// TIA Portal project "SelecaoProjeto" (V15)

(* hardware
DEVICE "S7-1200 station_1"  S7-1200 Station
   slot 0: "Rack_0"  S7-1200 Rack  Rack  V1.0
   slot 1: "PLC_1"  CPU 1214C DC/DC/DC  6ES7 214-1AG40-0XB0  V4.2
   slot 2: "DI 8x24VDC_1"  SM 1221 DI8 x 24VDC  6ES7 221-1BF30-0XB0  V1.0
*)

// ===== PLC "PLC_1"  CPU 1214C DC/DC/DC =====

VAR_GLOBAL   // PLC tag table "Default tag table"
   "BtnStop" AT %I0.0 : Bool;
   "BtnStart" AT %I0.1 : Bool;
   "S2Capacitivo" AT %I0.2 : Bool;
   "S1Indutivo" AT %I0.3 : Bool;
   "S3Pequeno" AT %I0.4 : Bool;
   "S4Medio" AT %I0.5 : Bool;
   "S5Grande" AT %I0.6 : Bool;
   "Resetar defeito" AT %I0.7 : Bool;
   "S6_FimDeCurso" AT %I1.0 : Bool;
   "Reed_Switch1" AT %I1.1 : Bool;
   "Reed_Switch2" AT %I1.2 : Bool;
   "Reed_Switch3" AT %I1.3 : Bool;
   "SnOtico_Grande" AT %I1.4 : Bool;
   "SnOtico_Medio" AT %I1.5 : Bool;
   "SnOtico_Pequeno" AT %I8.0 : Bool;
   "Motor1" AT %Q0.1 : Bool;
   "LampadaDefeito" AT %Q0.2 : Bool;
   "Soleoneide1" AT %Q0.3 : Bool;
   "Soleoneide2" AT %Q0.4 : Bool;
   "Soleoneide3" AT %Q0.5 : Bool;
   "SemDefeito1" AT %M0.1 : Bool;
   "SemDefeito2" AT %M0.2 : Bool;
   "MotorPronto" AT %M0.4 : Bool;
   "S1acionado" AT %M0.5 : Bool;
   "S2Acionado" AT %M0.6 : Bool;
   "Metalico" AT %M1.0 : Bool;
   "NaoMetalico" AT %M1.1 : Bool;
   "Vazio" AT %M1.2 : Bool;
   "MotorSetado" AT %M0.7 : Bool;
   "S3Acionado" AT %M1.3 : Bool;
   "S4Acionado" AT %M1.4 : Bool;
   "S5Acionado" AT %M1.5 : Bool;
   "Grande" AT %M2.0 : Bool;
   "Medio" AT %M2.1 : Bool;
   "Pequeno" AT %M2.2 : Bool;
   "Vazio2" AT %M1.7 : Bool;
   "Sistema com defeito" AT %M3.0 : Bool;
   "Zera_Contagem" AT %M0.3 : Bool;
   "Rejeitado" AT %M4.0 : Bool;
   "Solenoide_Recuado" AT %M4.1 : Bool;
   "Contagem_Grande" AT %M4.2 : Bool;
   "Contagem_Media" AT %M4.3 : Bool;
   "Contagem_Pequena" AT %M4.4 : Bool;
END_VAR

// folder: System blocks/Program resources

DATA_BLOCK "IEC_Counter_0_DB"   // DB1
{ S7_Optimized_Access := 'TRUE' }
AUTHOR : Simatic
FAMILY : IEC
NAME : CNTR
VERSION : 1.0
// stored: InstanceOfName IEC_COUNTER
"IEC_COUNTER"
BEGIN
END_DATA_BLOCK

DATA_BLOCK "IEC_Counter_0_DB_2"   // DB3
{ S7_Optimized_Access := 'TRUE' }
AUTHOR : Simatic
FAMILY : IEC
NAME : CNTR
VERSION : 1.0
// stored: InstanceOfName IEC_COUNTER
"IEC_COUNTER"
BEGIN
END_DATA_BLOCK

DATA_BLOCK "IEC_Counter_0_DB_3"   // DB4
{ S7_Optimized_Access := 'TRUE' }
AUTHOR : Simatic
FAMILY : IEC
NAME : CNTR
VERSION : 1.0
// stored: InstanceOfName IEC_COUNTER
"IEC_COUNTER"
BEGIN
END_DATA_BLOCK

DATA_BLOCK "IEC_Counter_0_DB_4"   // DB5
{ S7_Optimized_Access := 'TRUE' }
AUTHOR : Simatic
FAMILY : IEC
NAME : CNTR
VERSION : 1.0
// stored: InstanceOfName IEC_COUNTER
"IEC_COUNTER"
BEGIN
END_DATA_BLOCK

// folder: (top level)

FUNCTION "Selecao" : Void   // FC1, LAD
{ S7_Optimized_Access := 'TRUE' }
VERSION : 0.1
// Projeto Separação de peças
BEGIN

REGION Network 1
   // Setar Motor
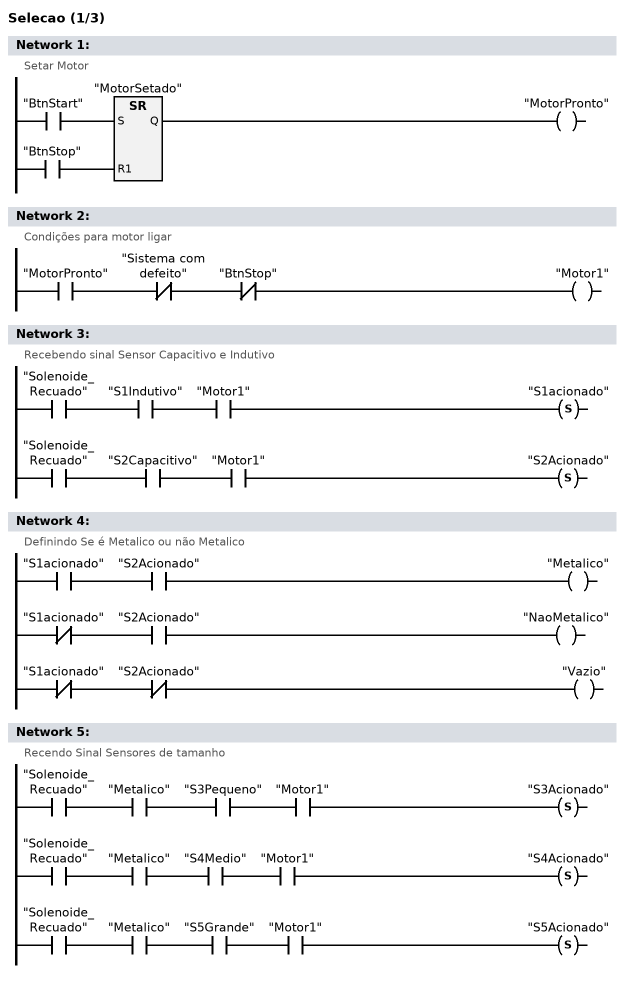
   RUNG wire#powerrail
      Contact( "BtnStart" )
      S_SR(operand := "MotorSetado", r1 := wire#w1)
      Coil( "MotorPronto" )
   END_RUNG
   RUNG wire#powerrail
      Contact( "BtnStop" )
   END_RUNG wire#w1
   // the same network as SCL:
   IF "BtnStart" THEN
       "MotorSetado" := TRUE;   // SR flip-flop
   END_IF;
   IF "BtnStop" THEN "MotorSetado" := FALSE; END_IF;
   "MotorPronto" := "MotorSetado";
END_REGION

REGION Network 2
   // Condições para motor ligar
   RUNG wire#powerrail
      Contact( "MotorPronto" )
      I_Contact( "Sistema com defeito" )
      I_Contact( "BtnStop" )
      Coil( "Motor1" )
   END_RUNG
   // the same network as SCL:
   "Motor1" := "MotorPronto" AND NOT "Sistema com defeito" AND NOT "BtnStop";
END_REGION

REGION Network 3
   // Recebendo sinal Sensor Capacitivo e Indutivo
   RUNG wire#powerrail
      Contact( "Solenoide_Recuado" )
      Contact( "S1Indutivo" )
      Contact( "Motor1" )
      S_Coil( "S1acionado" )
   END_RUNG
   RUNG wire#powerrail
      Contact( "Solenoide_Recuado" )
      Contact( "S2Capacitivo" )
      Contact( "Motor1" )
      S_Coil( "S2Acionado" )
   END_RUNG
   // the same network as SCL:
   IF "Solenoide_Recuado" AND "S1Indutivo" AND "Motor1" THEN "S1acionado" := TRUE; END_IF;
   IF "Solenoide_Recuado" AND "S2Capacitivo" AND "Motor1" THEN "S2Acionado" := TRUE; END_IF;
END_REGION

REGION Network 4
   // Definindo Se é Metalico ou não Metalico
   RUNG wire#powerrail
      Contact( "S1acionado" )
      Contact( "S2Acionado" )
      Coil( "Metalico" )
   END_RUNG
   RUNG wire#powerrail
      I_Contact( "S1acionado" )
      Contact( "S2Acionado" )
      Coil( "NaoMetalico" )
   END_RUNG
   RUNG wire#powerrail
      I_Contact( "S1acionado" )
      I_Contact( "S2Acionado" )
      Coil( "Vazio" )
   END_RUNG
   // the same network as SCL:
   "Metalico" := "S1acionado" AND "S2Acionado";
   "NaoMetalico" := NOT "S1acionado" AND "S2Acionado";
   "Vazio" := NOT "S1acionado" AND NOT "S2Acionado";
END_REGION

REGION Network 5
   // Recendo Sinal Sensores de tamanho
   RUNG wire#powerrail
      Contact( "Solenoide_Recuado" )
      Contact( "Metalico" )
      Contact( "S3Pequeno" )
      Contact( "Motor1" )
      S_Coil( "S3Acionado" )
   END_RUNG
   RUNG wire#powerrail
      Contact( "Solenoide_Recuado" )
      Contact( "Metalico" )
      Contact( "S4Medio" )
      Contact( "Motor1" )
      S_Coil( "S4Acionado" )
   END_RUNG
   RUNG wire#powerrail
      Contact( "Solenoide_Recuado" )
      Contact( "Metalico" )
      Contact( "S5Grande" )
      Contact( "Motor1" )
      S_Coil( "S5Acionado" )
   END_RUNG
   // the same network as SCL:
   IF "Solenoide_Recuado" AND "Metalico" AND "S3Pequeno" AND "Motor1" THEN "S3Acionado" := TRUE; END_IF;
   IF "Solenoide_Recuado" AND "Metalico" AND "S4Medio" AND "Motor1" THEN "S4Acionado" := TRUE; END_IF;
   IF "Solenoide_Recuado" AND "Metalico" AND "S5Grande" AND "Motor1" THEN "S5Acionado" := TRUE; END_IF;
END_REGION

REGION Network 6
   // Definindo se sensor é grande, medio ou pequeno
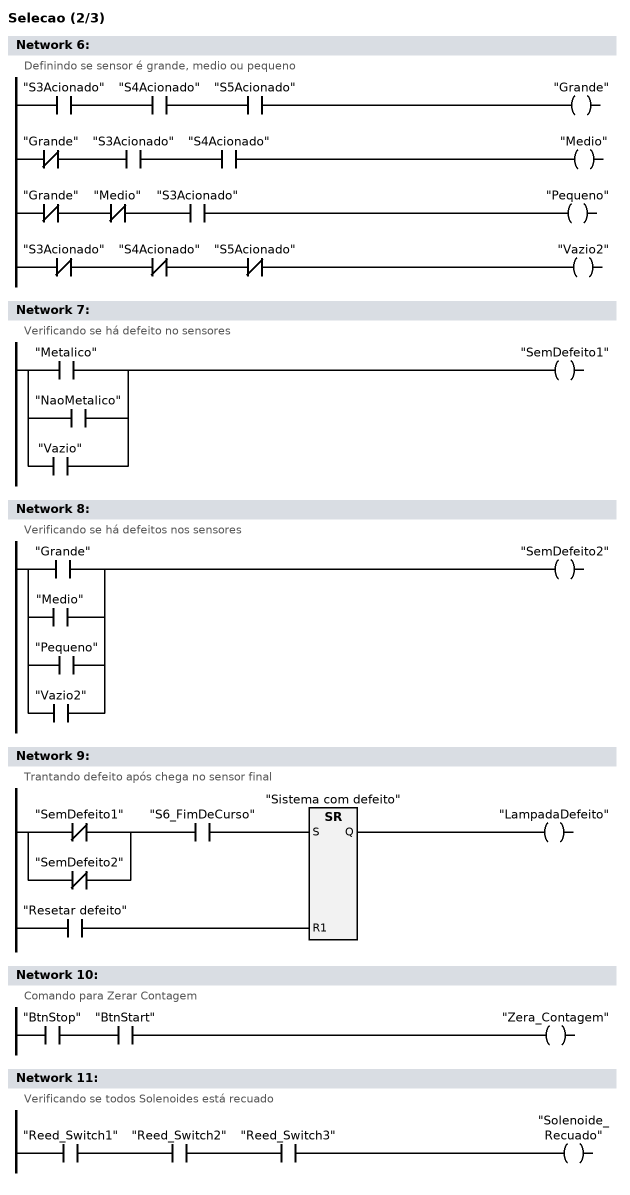
   RUNG wire#powerrail
      Contact( "S3Acionado" )
      Contact( "S4Acionado" )
      Contact( "S5Acionado" )
      Coil( "Grande" )
   END_RUNG
   RUNG wire#powerrail
      I_Contact( "Grande" )
      Contact( "S3Acionado" )
      Contact( "S4Acionado" )
      Coil( "Medio" )
   END_RUNG
   RUNG wire#powerrail
      I_Contact( "Grande" )
      I_Contact( "Medio" )
      Contact( "S3Acionado" )
      Coil( "Pequeno" )
   END_RUNG
   RUNG wire#powerrail
      I_Contact( "S3Acionado" )
      I_Contact( "S4Acionado" )
      I_Contact( "S5Acionado" )
      Coil( "Vazio2" )
   END_RUNG
   // the same network as SCL:
   "Grande" := "S3Acionado" AND "S4Acionado" AND "S5Acionado";
   "Medio" := NOT "Grande" AND "S3Acionado" AND "S4Acionado";
   "Pequeno" := NOT "Grande" AND NOT "Medio" AND "S3Acionado";
   "Vazio2" := NOT "S3Acionado" AND NOT "S4Acionado" AND NOT "S5Acionado";
END_REGION

REGION Network 7
   // Verificando se há defeito no sensores
   RUNG wire#powerrail
      Contact( "Metalico" )
      wire#w1
      Coil( "SemDefeito1" )
   END_RUNG
   RUNG wire#powerrail
      Contact( "NaoMetalico" )
   END_RUNG wire#w1
   RUNG wire#powerrail
      Contact( "Vazio" )
   END_RUNG wire#w1
   // the same network as SCL:
   "SemDefeito1" := "Metalico" OR "NaoMetalico" OR "Vazio";
END_REGION

REGION Network 8
   // Verificando se há defeitos nos sensores
   RUNG wire#powerrail
      Contact( "Grande" )
      wire#w1
      Coil( "SemDefeito2" )
   END_RUNG
   RUNG wire#powerrail
      Contact( "Medio" )
   END_RUNG wire#w1
   RUNG wire#powerrail
      Contact( "Pequeno" )
   END_RUNG wire#w1
   RUNG wire#powerrail
      Contact( "Vazio2" )
   END_RUNG wire#w1
   // the same network as SCL:
   "SemDefeito2" := "Grande" OR "Medio" OR "Pequeno" OR "Vazio2";
END_REGION

REGION Network 9
   // Trantando defeito após chega no sensor final
   RUNG wire#powerrail
      I_Contact( "SemDefeito1" )
      wire#w1
      Contact( "S6_FimDeCurso" )
      S_SR(operand := "Sistema com defeito", r1 := wire#w2)
      Coil( "LampadaDefeito" )
   END_RUNG
   RUNG wire#powerrail
      I_Contact( "SemDefeito2" )
   END_RUNG wire#w1
   RUNG wire#powerrail
      Contact( "Resetar defeito" )
   END_RUNG wire#w2
   // the same network as SCL:
   IF (NOT "SemDefeito1" OR NOT "SemDefeito2") AND "S6_FimDeCurso" THEN
       "Sistema com defeito" := TRUE;   // SR flip-flop
   END_IF;
   IF "Resetar defeito" THEN "Sistema com defeito" := FALSE; END_IF;
   "LampadaDefeito" := "Sistema com defeito";
END_REGION

REGION Network 10
   // Comando para Zerar Contagem
   RUNG wire#powerrail
      Contact( "BtnStop" )
      Contact( "BtnStart" )
      Coil( "Zera_Contagem" )
   END_RUNG
   // the same network as SCL:
   "Zera_Contagem" := "BtnStop" AND "BtnStart";
END_REGION

REGION Network 11
   // Verificando se todos Solenoides está recuado
   RUNG wire#powerrail
      Contact( "Reed_Switch1" )
      Contact( "Reed_Switch2" )
      Contact( "Reed_Switch3" )
      Coil( "Solenoide_Recuado" )
   END_RUNG
   // the same network as SCL:
   "Solenoide_Recuado" := "Reed_Switch1" AND "Reed_Switch2" AND "Reed_Switch3";
END_REGION

REGION Network 12
   // Acionando Soleoneides
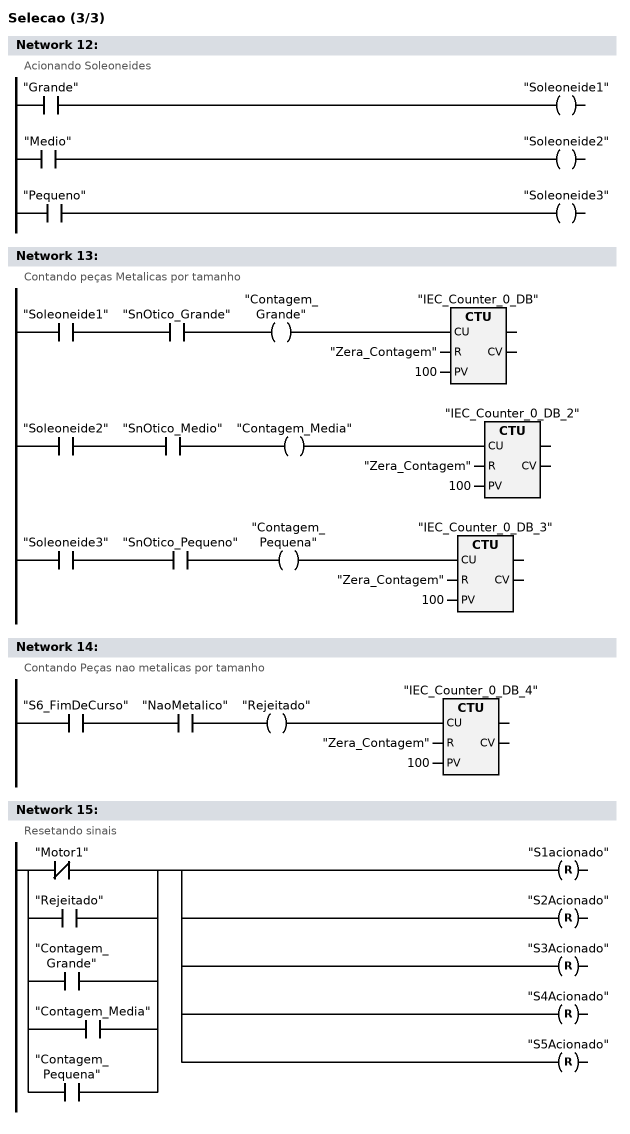
   RUNG wire#powerrail
      Contact( "Grande" )
      Coil( "Soleoneide1" )
   END_RUNG
   RUNG wire#powerrail
      Contact( "Medio" )
      Coil( "Soleoneide2" )
   END_RUNG
   RUNG wire#powerrail
      Contact( "Pequeno" )
      Coil( "Soleoneide3" )
   END_RUNG
   // the same network as SCL:
   "Soleoneide1" := "Grande";
   "Soleoneide2" := "Medio";
   "Soleoneide3" := "Pequeno";
END_REGION

REGION Network 13
   // Contando peças Metalicas por tamanho
   "Contagem_Grande" := "Soleoneide1" AND "SnOtico_Grande";
   "IEC_Counter_0_DB".CTU(CU := "Contagem_Grande", R := "Zera_Contagem", PV := 100);
   "Contagem_Media" := "Soleoneide2" AND "SnOtico_Medio";
   "IEC_Counter_0_DB_2".CTU(CU := "Contagem_Media", R := "Zera_Contagem", PV := 100);
   "Contagem_Pequena" := "Soleoneide3" AND "SnOtico_Pequeno";
   "IEC_Counter_0_DB_3".CTU(CU := "Contagem_Pequena", R := "Zera_Contagem", PV := 100);
END_REGION

REGION Network 14
   // Contando Peças nao metalicas por tamanho
   "Rejeitado" := "S6_FimDeCurso" AND "NaoMetalico";
   "IEC_Counter_0_DB_4".CTU(CU := "Rejeitado", R := "Zera_Contagem", PV := 100);
END_REGION

REGION Network 15
   // Resetando sinais
   RUNG wire#powerrail
      I_Contact( "Motor1" )
      wire#w1
      R_Coil( "S1acionado" )
   END_RUNG
   RUNG wire#powerrail
      Contact( "Rejeitado" )
   END_RUNG wire#w1
   RUNG wire#powerrail
      Contact( "Contagem_Grande" )
   END_RUNG wire#w1
   RUNG wire#powerrail
      Contact( "Contagem_Media" )
   END_RUNG wire#w1
   RUNG wire#powerrail
      Contact( "Contagem_Pequena" )
   END_RUNG wire#w1
   RUNG wire#w1
      R_Coil( "S2Acionado" )
   END_RUNG
   RUNG wire#w1
      R_Coil( "S3Acionado" )
   END_RUNG
   RUNG wire#w1
      R_Coil( "S4Acionado" )
   END_RUNG
   RUNG wire#w1
      R_Coil( "S5Acionado" )
   END_RUNG
   // the same network as SCL:
   IF NOT "Motor1" OR "Rejeitado" OR "Contagem_Grande" OR "Contagem_Media" OR "Contagem_Pequena" THEN
       "S1acionado" := FALSE;
       "S2Acionado" := FALSE;
       "S3Acionado" := FALSE;
       "S4Acionado" := FALSE;
       "S5Acionado" := FALSE;
   END_IF;
END_REGION
END_FUNCTION

ORGANIZATION_BLOCK "Main"   // OB1, LAD, ProgramCycle
TITLE = "Main Program Sweep (Cycle)"
{ S7_Optimized_Access := 'TRUE' }
VERSION : 0.1
   VAR_INPUT
      Initial_Call : Bool;   // Initial call of this OB
      Remanence : Bool;   // =True, if remanent data are available
   END_VAR
BEGIN

REGION Network 1
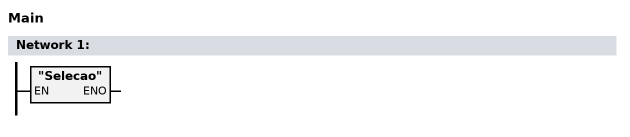
   RUNG wire#powerrail
      "Selecao"()
   END_RUNG
   // the same network as SCL:
   "Selecao"();
END_REGION
END_ORGANIZATION_BLOCK